SUBAPPLICATION RampLimitFS_TO_logiBUS_QDA_PWM_OPC (* Ein PWM-Kanal (0-100% Duty): VT-Zahlenfeld+Balkengrafik+6 Ramp-Tasten, physischer PWM-Ausgang, OPC-UA Publish/Subscribe (generisch, ein Kanal) *)
  (* Standard: 61499-2; Description: Copyright (c) 2026 Meisterschulen am Ostbahnhof This program and the accompanying materials are made available under the terms of the Eclipse Public License 2.0 which is available at https://www.eclipse.org/legal/epl-2.0/ SPDX-License-Identifier: EPL-2.0 *)
  (* Version 1.0, 2026-08-28, Franz Höpfinger, Meisterschulen am Ostbahnhof, initial API and implementation and/or initial documentation *)
  PACKAGE MyLib::sys;
  IMPORT isobus::UT::Q::const::IDs::ID_NULL;
  IMPORT logiBUS::io::DQ::logiBUS_DO;
  IMPORT logiBUS::io::DQ::logiBUS_DO_S;
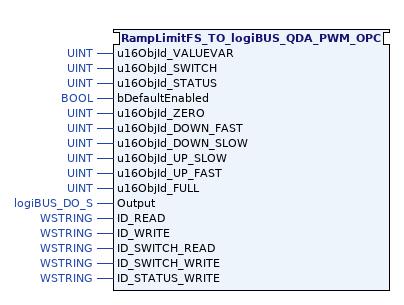
  VAR_INPUT
    u16ObjId_VALUEVAR : UINT := ID_NULL; (* Object ID CNumberVariable (Prozent 0-100, gemeinsam gebunden an Balkengrafik und CInputNumber-Anzeige) *)
    u16ObjId_SWITCH : UINT := ID_NULL; (* Object ID Kanal-Ein/Aus-Taste (Klick togglet Enable) *)
    u16ObjId_STATUS : UINT := ID_NULL; (* Object ID Status-Anzeige (Hintergrundfarbe Weiss=Kanal deaktiviert / Gruen=aktiv+logiBUS_QD_PWM.QO TRUE / Rot=aktiv+QO FALSE, Stoerung) *)
    bDefaultEnabled : BOOL; (* Kanal-Zustand beim Start: TRUE=aktiv (Kanaele 1-8), FALSE=inaktiv (Kanaele 9-12, da nur 8 Kanaele pro Controller gleichzeitig verfuegbar sind) *)
    u16ObjId_ZERO : UINT := ID_NULL; (* Object ID Taste '0' (RampLimitFS.ZERO) *)
    u16ObjId_DOWN_FAST : UINT := ID_NULL; (* Object ID Taste '--' (RampLimitFS.DOWN_FAST, ~10%) *)
    u16ObjId_DOWN_SLOW : UINT := ID_NULL; (* Object ID Taste '-' (RampLimitFS.DOWN_SLOW, ~1%) *)
    u16ObjId_UP_SLOW : UINT := ID_NULL; (* Object ID Taste '+' (RampLimitFS.UP_SLOW, ~1%) *)
    u16ObjId_UP_FAST : UINT := ID_NULL; (* Object ID Taste '++' (RampLimitFS.UP_FAST, ~10%) *)
    u16ObjId_FULL : UINT := ID_NULL; (* Object ID Taste 'F' (RampLimitFS.FULL, 100%) *)
    Output : logiBUS::io::DQ::logiBUS_DO_S := logiBUS_DO::Invalid; (* Identify the PWM Output Output_Q1..Q12 *)
    ID_READ : WSTRING; (* Remote-Sollwert-Adresse (Prozent REAL, ACTION=SUBSCRIBE) *)
    ID_WRITE : WSTRING; (* Echo-Ruckmelde-Adresse (Prozent REAL, ACTION=PUBLISH) *)
    ID_SWITCH_READ : WSTRING; (* Remote-Schalter-Adresse (BOOL, ACTION=SUBSCRIBE, togglet Kanal-Enable wie ein Tastendruck) *)
    ID_SWITCH_WRITE : WSTRING; (* Echo-Ruckmelde-Adresse (BOOL, ACTION=PUBLISH, aktueller Kanal-Enable-Zustand) *)
    ID_STATUS_WRITE : WSTRING; (* Status-Ruckmelde-Adresse (BOOL, ACTION=PUBLISH, nur lesend, logiBUS_QD_PWM.QO) *)
  END_VAR
  (* Ja, gerechnet: 64255 × 8191 = 526.406.305. DINT (32-bit signed) geht bis 2.147.483.647 — der Zwischenwert nutzt nur ~25% des Wertebereichs, keine Überlauf-Gefahr. *)
  FBS
    NumericValue_Duty : isobus::UT::io::NumericValue::NumericValue_ID(QI := TRUE);
    F_DWORD_TO_UDINT_VT : iec61131::conversion::F_DWORD_TO_UDINT;
    F_UDINT_TO_DINT_VT : iec61131::conversion::F_UDINT_TO_DINT;
    AR_SUBSCRIBE_1 : adapter::net::AR_SUBSCRIBE_1(QI := TRUE);
    AR_R_TO_REAL_SUB : adapter::conversion::unidirectional::AR_R_TO_REAL;
    F_PERCENT_TO_FRACTION_SUB : logiBUS::signalprocessing::fieldbus::F_PERCENT_TO_FRACTION;
    RampLimitFS : eclipse4diac::signalprocessing::RampLimitFS(VAL_ZERO := DINT#0, SLOW := DINT#643, FAST := DINT#6426, VAL_FULL := DINT#64255);
    F_MUL_TO_PWM13BIT : iec61131::arithmetic::F_MUL(IN2 := DINT#8191);
    F_DIV_TO_PWM13BIT : iec61131::arithmetic::F_DIV(IN2 := DINT#64255);
    F_DINT_TO_DWORD_OUT : iec61131::conversion::F_DINT_TO_DWORD;
    logiBUS_QD_PWM : logiBUS::io::DQ::logiBUS_QD_PWM;
    F_DINT_TO_UDINT_DISP : iec61131::conversion::F_DINT_TO_UDINT;
    Q_NumericValue : isobus::UT::Q::Q_NumericValue;
    F_FRACTION_TO_PERCENT_PUB : logiBUS::signalprocessing::fieldbus::F_FRACTION_TO_PERCENT;
    AR_REAL_TO_R_PUB : adapter::conversion::unidirectional::AR_REAL_TO_R;
    AR_PUBLISH_1 : adapter::net::AR_PUBLISH_1(QI := TRUE);
    E_RS_PV : iec61499::events::E_RS;
    F_SEL_PV : iec61131::selection::F_SEL;
    F_MOVE : iec61131::selection::F_MOVE; {SET_ATTRIBUTE(DataType, DINT)}
    E_SPLIT_VT : iec61499::events::E_SPLIT_2;
    E_SPLIT_WEB : iec61499::events::E_SPLIT_2;
    E_MERGE_SEL : iec61499::events::E_MERGE_2;
    E_T_FF_SR_SWITCH : iec61499::events::E_T_FF_SR_SYM_INIT(QI := TRUE);
    AX_SUBSCRIBE_SWITCH : adapter::net::AX_SUBSCRIBE_1(QI := TRUE);
    AX_RF_TRIG_SWITCH : adapter::events::unidirectional::AX_RF_TRIG;
    AX_BOOL_TO_X_SWITCH : adapter::conversion::unidirectional::AX_BOOL_TO_X;
    AX_PUBLISH_SWITCH : adapter::net::AX_PUBLISH_1(QI := TRUE);
    AX_BOOL_TO_X_STATUS : adapter::conversion::unidirectional::AX_BOOL_TO_X;
    AX_PUBLISH_STATUS : adapter::net::AX_PUBLISH_1(QI := TRUE);
  END_FBS
  SUBAPPS
    F_PWM_PERCENT_TO_RAW : MyLib::sys::F_PWM_PERCENT_TO_RAW;
    F_PWM_RAW_TO_PERCENT : MyLib::sys::F_PWM_RAW_TO_PERCENT;
    Q_BackgroundColour_EnableOk_STATUS : MyLib::sys::Q_BackgroundColour_EnableOk;
    Ramp6Buttons : MyLib::sys::Ramp6Buttons;
  END_SUBAPPS
  EVENT_CONNECTIONS
    NumericValue_Duty.IND TO F_DWORD_TO_UDINT_VT.REQ;
    F_DWORD_TO_UDINT_VT.CNF TO F_UDINT_TO_DINT_VT.REQ;
    F_UDINT_TO_DINT_VT.CNF TO E_SPLIT_VT.EI;
    E_SPLIT_VT.EO1 TO E_RS_PV.R;
    E_SPLIT_VT.EO2 TO E_MERGE_SEL.EI1;
    AR_SUBSCRIBE_1.INITO TO AR_PUBLISH_1.INIT;
    AR_PUBLISH_1.INITO TO AX_SUBSCRIBE_SWITCH.INIT;
    AX_SUBSCRIBE_SWITCH.INITO TO AX_PUBLISH_SWITCH.INIT;
    AX_PUBLISH_SWITCH.INITO TO AX_PUBLISH_STATUS.INIT;
    AR_R_TO_REAL_SUB.CNF TO F_PERCENT_TO_FRACTION_SUB.REQ;
    F_PERCENT_TO_FRACTION_SUB.CNF TO F_PWM_PERCENT_TO_RAW.REQ;
    F_PWM_PERCENT_TO_RAW.CNF TO E_SPLIT_WEB.EI;
    E_SPLIT_WEB.EO1 TO E_RS_PV.S;
    E_SPLIT_WEB.EO2 TO E_MERGE_SEL.EI2;
    E_MERGE_SEL.EO TO F_SEL_PV.REQ;
    F_SEL_PV.CNF TO RampLimitFS.LOAD;
    E_T_FF_SR_SWITCH.EO TO logiBUS_QD_PWM.INIT;
    E_T_FF_SR_SWITCH.EO TO Q_BackgroundColour_EnableOk_STATUS.REQ;
    logiBUS_QD_PWM.INITO TO AX_BOOL_TO_X_SWITCH.REQ;
    logiBUS_QD_PWM.INITO TO Q_BackgroundColour_EnableOk_STATUS.REQ;
    logiBUS_QD_PWM.INITO TO AX_BOOL_TO_X_STATUS.REQ;
    RampLimitFS.CNF TO F_MUL_TO_PWM13BIT.REQ;
    F_MUL_TO_PWM13BIT.CNF TO F_MOVE.REQ;
    F_DIV_TO_PWM13BIT.CNF TO F_DINT_TO_DWORD_OUT.REQ;
    RampLimitFS.CNF TO F_DINT_TO_UDINT_DISP.REQ;
    RampLimitFS.CNF TO F_PWM_RAW_TO_PERCENT.REQ;
    F_DINT_TO_DWORD_OUT.CNF TO logiBUS_QD_PWM.REQ;
    F_DINT_TO_UDINT_DISP.CNF TO Q_NumericValue.REQ;
    F_PWM_RAW_TO_PERCENT.CNF TO F_FRACTION_TO_PERCENT_PUB.REQ;
    F_FRACTION_TO_PERCENT_PUB.CNF TO AR_REAL_TO_R_PUB.REQ;
    F_MOVE.CNF TO F_DIV_TO_PWM13BIT.REQ;
    Ramp6Buttons.IND_SWITCH TO E_T_FF_SR_SWITCH.CLK;
    Ramp6Buttons.IND_ZERO TO RampLimitFS.ZERO;
    Ramp6Buttons.IND_UP_SLOW TO RampLimitFS.UP_SLOW;
    Ramp6Buttons.IND_UP_FAST TO RampLimitFS.UP_FAST;
    Ramp6Buttons.IND_DOWN_SLOW TO RampLimitFS.DOWN_SLOW;
    Ramp6Buttons.IND_DOWN_FAST TO RampLimitFS.DOWN_FAST;
    Ramp6Buttons.IND_FULL TO RampLimitFS.FULL;
    AX_RF_TRIG_SWITCH.ER TO E_T_FF_SR_SWITCH.S;
    AX_RF_TRIG_SWITCH.EF TO E_T_FF_SR_SWITCH.R;
    AX_PUBLISH_STATUS.INITO TO E_T_FF_SR_SWITCH.INIT;
  END_CONNECTIONS
  DATA_CONNECTIONS
    u16ObjId_VALUEVAR TO NumericValue_Duty.u16ObjId;
    u16ObjId_VALUEVAR TO Q_NumericValue.u16ObjId;
    u16ObjId_STATUS TO Q_BackgroundColour_EnableOk_STATUS.u16ObjId;
    E_T_FF_SR_SWITCH.Q TO logiBUS_QD_PWM.QI;
    E_T_FF_SR_SWITCH.Q TO Q_BackgroundColour_EnableOk_STATUS.bEnable;
    logiBUS_QD_PWM.QO TO Q_BackgroundColour_EnableOk_STATUS.bOk;
    Output TO logiBUS_QD_PWM.Output;
    ID_READ TO AR_SUBSCRIBE_1.ID;
    ID_WRITE TO AR_PUBLISH_1.ID;
    ID_SWITCH_READ TO AX_SUBSCRIBE_SWITCH.ID;
    ID_SWITCH_WRITE TO AX_PUBLISH_SWITCH.ID;
    ID_STATUS_WRITE TO AX_PUBLISH_STATUS.ID;
    E_T_FF_SR_SWITCH.Q TO AX_BOOL_TO_X_SWITCH.OUT;
    logiBUS_QD_PWM.QO TO AX_BOOL_TO_X_STATUS.OUT;
    NumericValue_Duty.IN TO F_DWORD_TO_UDINT_VT.IN;
    F_DWORD_TO_UDINT_VT.OUT TO F_UDINT_TO_DINT_VT.IN;
    F_UDINT_TO_DINT_VT.OUT TO F_SEL_PV.IN0;
    AR_R_TO_REAL_SUB.IN TO F_PERCENT_TO_FRACTION_SUB.rPercent;
    F_PERCENT_TO_FRACTION_SUB.rFraction TO F_PWM_PERCENT_TO_RAW.IN;
    F_PWM_PERCENT_TO_RAW.OUT TO F_SEL_PV.IN1;
    E_RS_PV.Q TO F_SEL_PV.G;
    F_SEL_PV.OUT TO RampLimitFS.PV;
    RampLimitFS.OUT TO F_MUL_TO_PWM13BIT.IN1;
    F_MUL_TO_PWM13BIT.OUT TO F_MOVE.IN;
    F_DIV_TO_PWM13BIT.OUT TO F_DINT_TO_DWORD_OUT.IN;
    RampLimitFS.OUT TO F_DINT_TO_UDINT_DISP.IN;
    RampLimitFS.OUT TO F_PWM_RAW_TO_PERCENT.IN;
    F_DINT_TO_DWORD_OUT.OUT TO logiBUS_QD_PWM.OUT;
    F_DINT_TO_UDINT_DISP.OUT TO Q_NumericValue.u32NewValue;
    F_PWM_RAW_TO_PERCENT.OUT TO F_FRACTION_TO_PERCENT_PUB.rFraction;
    F_FRACTION_TO_PERCENT_PUB.rPercent TO AR_REAL_TO_R_PUB.OUT;
    F_MOVE.OUT TO F_DIV_TO_PWM13BIT.IN1;
    u16ObjId_SWITCH TO Ramp6Buttons.u16ObjId_SWITCH;
    u16ObjId_ZERO TO Ramp6Buttons.u16ObjId_ZERO;
    u16ObjId_UP_SLOW TO Ramp6Buttons.u16ObjId_UP_SLOW;
    u16ObjId_UP_FAST TO Ramp6Buttons.u16ObjId_UP_FAST;
    u16ObjId_DOWN_SLOW TO Ramp6Buttons.u16ObjId_DOWN_SLOW;
    u16ObjId_DOWN_FAST TO Ramp6Buttons.u16ObjId_DOWN_FAST;
    u16ObjId_FULL TO Ramp6Buttons.u16ObjId_FULL;
    bDefaultEnabled TO E_T_FF_SR_SWITCH.Q_INIT;
  END_CONNECTIONS
  ADAPTER_CONNECTIONS
    AR_SUBSCRIBE_1.OUT TO AR_R_TO_REAL_SUB.AR_IN;
    AX_SUBSCRIBE_SWITCH.OUT TO AX_RF_TRIG_SWITCH.QI;
    AR_REAL_TO_R_PUB.AR_OUT TO AR_PUBLISH_1.IN;
    AX_BOOL_TO_X_SWITCH.AX_OUT TO AX_PUBLISH_SWITCH.IN;
    AX_BOOL_TO_X_STATUS.AX_OUT TO AX_PUBLISH_STATUS.IN;
  END_CONNECTIONS
END_SUBAPPLICATION
